PROGRAM SummeGewichte
VAR
END_VAR

END_PROGRAM

(* stored: Version 1.1.0.1, ProductVersion 3.1.4018.5
   POU SummeGewichte: Id {ff6fce1c-ae1c-4f56-8146-d5e0b11ba922}, SpecialFunc None *)
